{attribute 'GeneratedUsingTerminal: EL1252-0000-0018'}
{attribute addProperty BoxType "EL1252-0000-0018"}
{attribute addProperty Id "Status1AT %I*USINT1Status2AT %I*USINT1LatchPos1AT %I*ULINT8LatchNeg1AT %I*ULINT8LatchPos2AT %I*ULINT8LatchNeg2AT %I*ULINT8"}
{attribute addProperty CRC "968719484"}
{attribute addProperty Size "34"}
TYPE Latch_39BD7C7C :
STRUCT
	{attribute addProperty Name "Status1"}
	Status1 AT %I* : USINT;
	{attribute addProperty Name "Status2"}
	Status2 AT %I* : USINT;
	{attribute addProperty Name "LatchPos1"}
	LatchPos1 AT %I* : ULINT;
	{attribute addProperty Name "LatchNeg1"}
	LatchNeg1 AT %I* : ULINT;
	{attribute addProperty Name "LatchPos2"}
	LatchPos2 AT %I* : ULINT;
	{attribute addProperty Name "LatchNeg2"}
	LatchNeg2 AT %I* : ULINT;
END_STRUCT
END_TYPE

(* stored: Version 1.2.0.0, ProductVersion 3.1.4024.9
   DUT Latch_39BD7C7C: Id {f58c20f1-1997-4a1c-b901-35f1e9226c48} *)
